// FICTIONAL ENGINEERING PROJECT — NOT FOR CONSTRUCTION
DATA_BLOCK "DB_CellMain"
{ S7_Optimized_Access := 'TRUE' }
VERSION : 0.1
NON_RETAIN
   "FB_CellMain"
BEGIN
END_DATA_BLOCK
